TYPE ST_Event :
STRUCT
	eEventTypes: E_EventType;
	eEventSeverity: TcEventSeverity;
	eEventIdentity: UDINT;
	eEventText: STRING(255);
	dtTimestamp: DATE_AND_TIME;	
END_STRUCT
END_TYPE

(* stored: Version 1.1.0.1, ProductVersion 3.1.4024.12
   DUT ST_Event: Id {d0828339-bc4a-4c30-8f44-adfb2e0669ce} *)
